# EPICS substitutions: 3-6/GalilTestApp/Db/galil_coordinate_systems.substitutions
# Description:
# Coordinate systems substitution file.
#
# This library is free software; you can redistribute it and/or
# modify it under the terms of the GNU Lesser General Public
# Licence as published by the Free Software Foundation; either
# version 2.1 of the Licence, or (at your option) any later version.
#
# This library is distributed in the hope that it will be useful,
# but WITHOUT ANY WARRANTY; without even the implied warranty of
# MERCHANTABILITY or FITNESS FOR A PARTICULAR PURPOSE.  See the GNU
# Lesser General Public Licence for more details.
#
# You should have received a copy of the GNU Lesser General Public
# Licence along with this library; if not, write to the Free Software
# Foundation, Inc., 51 Franklin St, Fifth Floor, Boston, MA 02110-1301 USA.
#
# Contact details:
# Mark Clift
# email: padmoz@tpg.com.au

# Coordinate system status
#
# R    - Record Name
# ADDR - Hardware port to read
# SCAN - Scan period for monitor records

file "$(GALIL)/GalilSup/Db/galil_coordinate_system.template"
{
pattern { R,    ADDR,  SCAN         }

        { "S",  "0",   ".1 second"  }
        { "T",  "1",   ".1 second"  }
}

# end
